(* CODESYS project stopwatch_level.library
   Author: Víctor Durán Muñoz
   Placeholder: library_StopWatch_Level
   Title: library_StopWatch_Level
   Version: 1.0
   Company: Automatizaciones Adegar

Project tree, tasks and I/O mapping:
  libraries: Tc2_Standard, * (Beckhoff Automation GmbH); Tc2_System, * (Beckhoff Automation GmbH); Tc3_Module, * (Beckhoff Automation GmbH)
  function block FB_StopWatch_Level [ST]
*)

// FB_StopWatch_Level
FUNCTION_BLOCK FB_StopWatch_Level
VAR_INPUT
	bSTART				:	BOOL;    // START
	bRESET				: 	BOOL;	// RESET
END_VAR
VAR_OUTPUT
	Elapsed_Time		: 	TIME;
END_VAR
VAR
	{attribute 'hide' := ''}
	Time_Count			: 	UDINT;
	{attribute 'hide' := ''}
	Current_CycleTime	: 	UDINT;
	{attribute 'hide' := ''}
	COUNT_TIME: BOOL 	:= 	FALSE;
	{attribute 'hide' := ''}
	fbGetTaskIndex		: 	GETCURTASKINDEX;
END_VAR

// Count StopWatch.
IF bSTART AND NOT bRESET THEN
	fbGetTaskIndex();
	COUNT_TIME := TRUE;
	Current_CycleTime := TwinCAT_SystemInfoVarList._TaskInfo[fbGetTaskIndex.index].CycleTime (*100ns unit*);
END_IF

// Stop StopWatch.
IF NOT bSTART OR bRESET THEN
	COUNT_TIME := FALSE;
END_IF

// Reset StopWatch.
IF bRESET THEN	
	Time_Count := 0;
	Elapsed_Time := T#0MS;
END_IF

IF COUNT_TIME THEN
	Time_Count := Time_Count + Current_CycleTime;
	IF Time_Count > 10000 THEN		
		Elapsed_Time := Elapsed_Time + UDINT_TO_TIME(Time_Count/10000);
		Time_Count := 0;
	END_IF
END_IF

END_FUNCTION_BLOCK
